// TwinCAT 3 PLC project PLC
// ProgramVersion: 3.1.4024.0
// libraries:
//   SPT Base Types, * (Beckhoff Automation LLC)
//   SPT Components, * (Beckhoff Automation LLC)
//   SPT Motion Control, * (Beckhoff Automation LLC)
//   Tc2_Standard, * (Beckhoff Automation GmbH)
//   Tc2_System, * (Beckhoff Automation GmbH)
//   Tc3_Module, * (Beckhoff Automation GmbH)
// project tree:
//   / GlobalTextList.TcGTLO (not stored), PlcTask.TcTTO (not stored), Visualization Manager.TcVMO (not stored)
//   Modules/00 Machine/ Machine.TcPOU
//   POUs/ MAIN.TcPOU
//   VISUs/ Visualization.TcVIS
// real-time tasks:
//   TASK PlcTask: cycle T#10ms, priority 20, ADS port 350
// motion (NC):
// variable links:
//   PLC/PLC Instance <-> NC-Task 1 SAF/Axes/Axis 1
//     PlcTask Inputs/MAIN.Machine.AX5000.BasicAxis._Axis.NcToPlc <-> Outputs/ToPlc
//     PlcTask Outputs/MAIN.Machine.AX5000.BasicAxis._Axis.PlcToNc <-> Inputs/FromPlc

// ---- Modules/00 Machine/Machine.TcPOU
FUNCTION_BLOCK Machine EXTENDS FB_PackML_BaseModule
VAR
	AX5000	  : FB_Component_BasicAxis := (Name := 'AX 5000 Axis');
	SoE_Reset : FB_ResetRoutine_SoEDrive;
END_VAR

// Automatically enables and disables HMI control based on the PackML mode
METHOD PROTECTED HMIPermissions

// This method is called cyclically by CyclicLogic()
AllowHMIControl(TRUE);
END_METHOD

// Basic module initialization logic
METHOD PROTECTED Initialize : BOOL;
VAR
END_VAR

// This method is called by CyclicLogic() as required
Initialize := FALSE;
CASE DescendantSequenceState OF
	0:
		RegisterComponent(AX5000);
		AX5000.ResetMethod		:= SoE_Reset;
		DescendantSequenceState := DescendantSequenceState + 10;

	10:
		IF SUPER^.Initialize() THEN
			DescendantSequenceState := DescendantSequenceState + 10;
		END_IF

	20:
		Initialize := TRUE;
END_CASE
END_METHOD

END_FUNCTION_BLOCK

// ---- POUs/MAIN.TcPOU
PROGRAM MAIN
VAR
	Machine : Machine := (Name := 'Machine');
END_VAR

(*All sample code provided by Beckhoff Automation LLC are for illustrative purposes only and are provided “as is” and without any warranties, express or implied. Actual implementations in applications will vary significantly. Beckhoff Automation LLC shall have no liability for, and does not waive any rights in relation to, any code samples that it provides or the use of such code samples for any purpose.*)

(*
	The default reset for the FB_ComponentAxis is a CoE Reset which works on most Beckhoff drives.
	However, some drives like the AX5000 use SoE instead of CoE.
	The difference in hardware requires a different set of commands to be sent in order to preform a reset.
	Specificlly the SoE drives need to toggle IDN-99
	FB_ResetRoutine_SoEDrive and FB_ResetRoutine_CoEDrive are both defined within the SPT_MotionControl library.
	By default an instance of FB_ResetRoutine_CoEDrive is passed into the Property ResetMethod during Initialization
	In order to change this decalre an instance of FB_ResetRoutine_SoEDrive and pass the instance to 
	Axis.ResetMethod.
	Because the property accepts the I_MotionSequence interface and the FB_ResetRoutine_SoEDrive implements this interface,
	we can pass an instance of FB_ResetRoutine_SoEDrive to the property. This is known as the strategy pattern, and it is also used 
	for the HomeMoethod and the ExternalSequence method.
	
	In this project open the Machine Module to see the declarations, and the Initialize method to see the assignment of the ResetMethod property.

*)

//This is for debug only and should be removed
_AppInfo.KeepOutputsOnBP := TRUE;

//
Machine.CyclicLogic();

END_PROGRAM

// ---- VISUs/Visualization.TcVIS
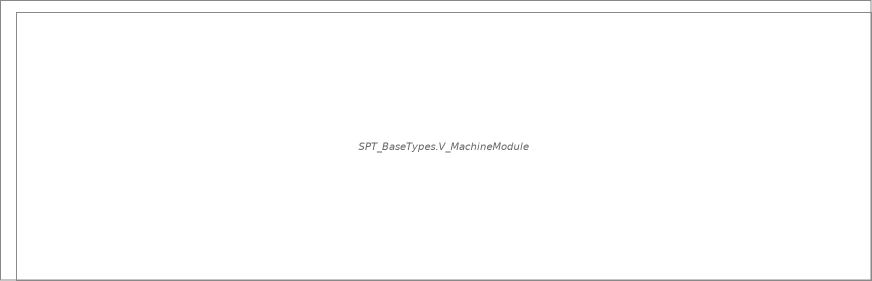
VISUALIZATION Visualization  // 872x281
    Frame (16,12 856x269)
        shows SPT_BaseTypes.V_MachineModule(HMI := MAIN.Machine.PackMLBaseModule_HMI)
END_VISUALIZATION
